// TIA Portal V21 export
DATA_BLOCK "BasicPosControl"   // DB7
// stored: InstanceOfName BasicPosControl_1, OfSystemLibElement BasicPosControl, OfSystemLibVersion 3.1
BasicPosControl_1   // technology object, version 3.1
   // VAR_INPUT
   //    ModePos : Int;
   //    EnableAxis : Bool;
   //    CancelTraversing : Bool;
   //    IntermediateStop : Bool;
   //    Positive : Bool;
   //    Negative : Bool;
   //    Jog1 : Bool;
   //    Jog2 : Bool;
   //    FlyRef : Bool;
   //    AckError : Bool;
   //    ExecuteMode : Bool;
   //    Position : LReal;
   //    Velocity : LReal;
   //    OverV : Int;
   //    OverAcc : Int;
   //    OverDec : Int;
   //    HomePosition : LReal;
   //    ConfigEPos : DWord;
   //    UserSetPZD : Word;
   // END_VAR
   // VAR_OUTPUT
   //    AxisEnabled : Bool;
   //    AxisPosOk : Bool;
   //    AxisSpFixed : Bool;
   //    AxisRef : Bool;
   //    AxisWarn : Bool;
   //    AxisError : Bool;
   //    Lockout : Bool;
   //    ActVelocity : LReal;
   //    ActPosition : LReal;
   //    ActMode : Int;
   //    EPosZSW1 : Word;
   //    EPosZSW2 : Word;
   //    ActWarn : Word;
   //    ActFault : Word;
   //    Error : Bool;
   //    Status : Word;
   //    DiagID : Word;
   //    UserReceivePZD : Word;
   // END_VAR
   // VAR
   //    sbOff1Edge : Bool;
   //    sbOff1 : Bool;
   //    sbExecuteEdge : Bool;
   //    sbExecute : Bool;
   //    sbRefTypEdge : Bool;
   //    sbRefTyp : Bool;
   //    sbMdiStart : Bool;
   //    sbMdiStartEdge : Bool;
   //    sbRefStart : Bool;
   //    sbJogInc : Bool;
   //    sbReady : Bool;
   //    sbIOp : Bool;
   //    sbAccel : Bool;
   //    sbDecel : Bool;
   //    sbAlarm : Bool;
   //    sbFault : Bool;
   //    sbFWD : Bool;
   //    sbBWD : Bool;
   //    sbBusy : Bool;
   //    swStatus : Word;
   //    swEPosZSW1 : Word;
   //    swEPosZSW2 : Word;
   //    siExecuteCyc : Int;
   //    siRefTypCyc : Int;
   //    siJogIncCyc : Int;
   //    siMdiStartCyc : Int;
   //    siRefActRetry : Int;
   //    siModePos : Int;
   //    siModePosMax : Int;
   //    siModePosMax_3rdGen : Int;
   //    siCycWait : Int;
   //    siRetryMax : Int;
   //    sbModePos : Bool;
   //    STW1 : Word;
   //    EPosSTW1 : Word;
   //    EPosSTW2 : Word;
   //    STW2 : Word;
   //    OverrideV : Word;
   //    PositionSP : DWord;
   //    VelocitySP : DWord;
   //    OverrideA : Word;
   //    OverrideA_DW : DWord;
   //    OverrideD : Word;
   //    OverrideD_DW : DWord;
   //    SendPZD12 : Word;
   //    ZSW1 : Word;
   //    EPosZSW3 : Word;
   //    EPosZSW4 : Word;
   //    ZSW2 : Word;
   //    NotUsed : Word;
   //    RES : DWord;
   //    REF_COORDINATE_DW : DWord;
   //    PositionAV : DWord;
   //    VelocityAV : DWord;
   //    ErrNr : Word;
   //    WarnNr : Word;
   //    ReceivePZD12 : Word;
   //    HWIDSTW : HW_IO := 280;
   //    HWIDZSW : HW_IO := 280;
   //    srResolutionFactor : LReal;
   //    srVelocityFactor : LReal;
   //    srNIST_BFactor : LReal := 2.79396772384644E-05;
   //    sDriveTelNo : Int;
   // END_VAR
BEGIN
END_DATA_BLOCK
